FUNCTION FindMinMax : REAL
VAR_INPUT
END_VAR
VAR_IN_OUT
	aRefArray : ARRAY[1..20] OF REAL;
END_VAR
VAR
	nIterator : INT;
END_VAR
VAR_OUTPUT
	fMinWeight : REAL ;
	fMaxWeight : REAL;
END_VAR


FOR nIterator := 2 TO 20 DO
	
	IF aRefArray[nIterator] = 0 THEN
		CONTINUE;
	END_IF
	
	IF fMinWeight = 0 THEN
		fMinWeight := aRefArray[nIterator];
		fMaxWeight := aRefArray[nIterator];
	END_IF
	
	IF aRefArray[nIterator] < fMinWeight THEN
		fMinWeight := aRefArray[nIterator];
	END_IF
	
	IF aRefArray[nIterator] > fMaxWeight THEN
		fMaxWeight := aRefArray[nIterator];
	END_IF
	
END_FOR

END_FUNCTION

(* stored: Version 1.1.0.1, ProductVersion 3.1.4024.16
   POU FindMinMax: Id {0e96b9d6-e551-4295-95b3-fc614fdf8692}, SpecialFunc None *)
